{attribute 'qualified_only'}
VAR_GLOBAL
	//OUTPUTS
	Prop_Valve AT %Q* : INT; 
	Pump_Start AT %Q* : BOOL;
	Pump_OL_Reset AT %Q* : BOOL;

	//INPUTS
	Process_Water_IN AT %I* : INT;
	Process_Water_OUT AT %I* : INT;
	Process_Water_FLOW AT %I* : INT;
	Process_Water_Setpoint : INT;
	Waterbath_Connection_Status AT %I* : UINT;
	Waterbath_System_Control AT %I* : BOOL;
	Pump_Fault AT %I* : BOOL;

	
	//System Variables
	Waterbath_StartwithSystem : BOOL;
	Waterbath_Start : BOOL;
	Waterbath_Running : BOOL;
	Waterbath_Local_Control : BOOL;
	
	//These are the HMI Variables after they are scaled correctly.
	Waterbath_SetPoint_Temp : REAL;
	Waterbath_Actual_Temp : REAL;
	Waterbath_Return_Temp : REAL;
	Waterbath_Flow_Rate : REAL;

	
	Waterbath_TempControl_Auto : BOOL;

	Waterbath_Delta_Temp : REAL;
	Waterbath_CalculatedBTULoss : REAL;
	
	Waterbath_Valve_Position_Percentage : REAL;
	
END_VAR

(* stored: Version 1.1.0.1, ProductVersion 3.1.4024.12
   GVL GVL_Waterbath: Id {4e0389f6-d444-475e-b034-359833017b6d} *)
